// TwinCAT 3 PLC project Tests_and_Samples
// ProgramVersion: 3.1.4023.0
// CompilerDefines: VISU_USEWSTRING
// libraries:
//   Tc2_Standard, * (Beckhoff Automation GmbH)
//   Tc2_System, * (Beckhoff Automation GmbH)
//   Tc3_BAR_Common, * (Beckhoff)
//   Tc3_Module, * (Beckhoff Automation GmbH)
// project tree:
//   / GlobalTextList.TcGTLO, GVL.TcGVL, PlcTask.TcTTO, Visualization Manager.TcVMO (not stored), VISU_TASK.TcTTO
//   GVLs/ Alarms.TcGVL
//   POUs/ AlarmSample.TcPOU, MAIN.TcPOU, TrendSample.TcPOU
//   VISUs/ AlarmsVisSample.TcVIS, TrendsSampleVis.TcVIS, vBrowser.TcVIS, Visualization.TcVIS
//   VISUs/Templates/ tAlarm.TcVIS
// (motion and I/O tree: see PLC project tc3_bar_common)
// real-time tasks:
//   TASK PlcTask: cycle T#10ms, priority 20, ADS port 350
//   TASK VISU_TASK: cycle T#50000us, priority 30, ADS port 351

CONFIGURATION Tests_and_Samples
    RESOURCE PLC ON TwinCAT3
        TASK PlcTask(INTERVAL := T#10ms, PRIORITY := 20);
        TASK VISU_TASK(INTERVAL := T#50000us, PRIORITY := 30);
        PROGRAM MAIN WITH PlcTask : MAIN;
        PROGRAM VisuElems_Visu_Prg WITH VISU_TASK : VisuElems.Visu_Prg;
    END_RESOURCE
END_CONFIGURATION

// ---- GVL.TcGVL
{attribute 'qualified_only'}
VAR_GLOBAL CONSTANT
END_VAR

// ---- GVLs/Alarms.TcGVL
{attribute 'qualified_only'}
VAR_GLOBAL
	SeriosAlarm: FB_Alarm := (AlarmInfo := (AlarmID := "LC224", Color := E_ALarmColors.E_Red, Description := "Серьезная тестовая авария", PossibleCause := "Оператор"));
	NotSeriosAlarm: FB_Alarm := (AlarmType := ALARMTYPE.Alarm_NoQuit, AlarmInfo := (AlarmID := "NQ105", Color := E_ALarmColors.E_Yellow, Description := "Ошибка, которую не нужно квитировать", PossibleCause := "Оператор"));
	SimpleWarning: FB_Alarm := (AlarmType := ALARMTYPE.Alarm_NoQuit, AlarmInfo := (AlarmID := "Wrn01", Color := E_ALarmColors.E_Green, Description := "Событие для записи в журнал", PossibleCause := "Оператор"));
END_VAR

// ---- POUs/MAIN.TcPOU
PROGRAM MAIN
VAR
	bBrowserStart: BOOL;
END_VAR

AlarmSample();// Пример работы с авариями

TrendSample();

END_PROGRAM

// ---- POUs/AlarmSample.TcPOU
PROGRAM AlarmSample
VAR

END_VAR

PRG_Alarms_Core();

END_PROGRAM

// ---- POUs/TrendSample.TcPOU
PROGRAM TrendSample
VAR
	VariableForTrend: REAL;
	t: REAL;
	VariableTrend: FB_TrendChanel := (MinimalValue := -1, MaximalValue := 1);
END_VAR

t:=t+0.01;
VariableForTrend:=SIN(t);
VariableTrend(InputData:= VariableForTrend);

END_PROGRAM

// ---- GlobalTextList.TcGTLO
TEXTLIST GlobalTextList
  789 = '\n\n%s'
  806 = '\n\nАварийное событие'
  101 = ' %s'
  133 = '%s'
  441 = 'PROFIT!?'
  574 = 'Аварийное событие'
  259 = 'История\nаварий'
  733 = 'История аварий'
  97 = 'Квитирование'
  906 = 'Квитирование\n этой аварии'
  227 = 'Квитирование\nвсех аварий'
  328 = 'Квитирование Аварии'
  893 = 'Квитирование этой аварии'
  440 = 'Название'
  618 = 'Название меню'
  740 = 'Пример\nаварий'
  504 = 'Пример\nТрендов'
  550 = 'Пример Аварий'
  641 = 'Пример ещё чего-то'
  12 = 'Пример трендов'
  306 = 'Пример Трендов'
  88 = 'Сброс'
  821 = 'Старт'
  100 = 'Стоп'
  839 = 'Текущие\n аварии'
  126 = 'Текущие\nаварии'
  188 = 'Текущие аварии'
  132 = 'Экран аварий'
END_TEXTLIST

// ---- VISUs/AlarmsVisSample.TcVIS
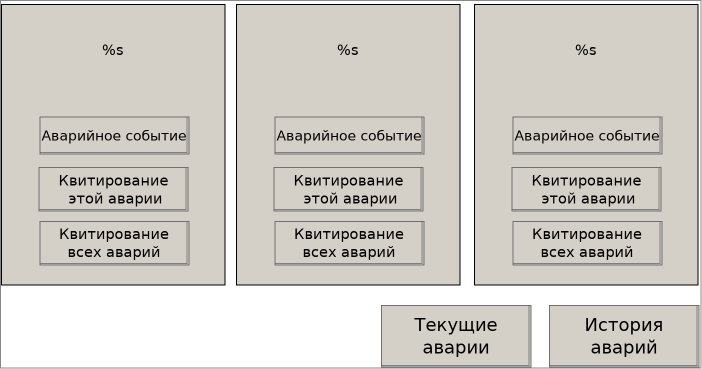
VISUALIZATION AlarmsVisSample  // 702x369
    Frame (1,4 226x283)
        shows tAlarm(alarm := Alarms.SeriosAlarm)
    Frame (236,4 226x283)
        shows tAlarm(alarm := Alarms.NotSeriosAlarm)
    Frame (474,4 226x283)
        shows tAlarm(alarm := Alarms.SimpleWarning)
    Button (381,305 150x62), "Текущие аварии"
        OnMouseClick: OpenDialog Dialog=Tc3_BAR_Common.Current_Alarms_dialog, OpenModal=True, OpenCentered=True
    Button (549,305 150x62), "История аварий"
        OnMouseClick: OpenDialog Dialog=Tc3_BAR_Common.History_Of_Alarms_dialog, OpenModal=True, OpenCentered=True
END_VISUALIZATION

// ---- VISUs/Templates/tAlarm.TcVIS
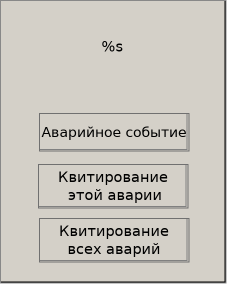
VISUALIZATION tAlarm  // 227x284
VAR_IN_OUT
	alarm: FB_Alarm;
END_VAR
    Rectangle (0,0 225x282), "%s", text variable: alarm.AlarmInfo.Description, colour toggle: Tc3_BAR_Common.LibAlarm.Blink and alarm.isActive
    Button (39,113 150x38), "Аварийное событие"
        toggle alarm.AlarmEvent
    Button (38,164 150x44), "Квитирование этой аварии"
        tap alarm.bQuitAlarm
    Button (39,218 150x44), "Квитирование всех аварий"
        tap Tc3_BAR_Common.LibAlarm.bLocalQuitAllAlarms
END_VISUALIZATION

// ---- VISUs/TrendsSampleVis.TcVIS
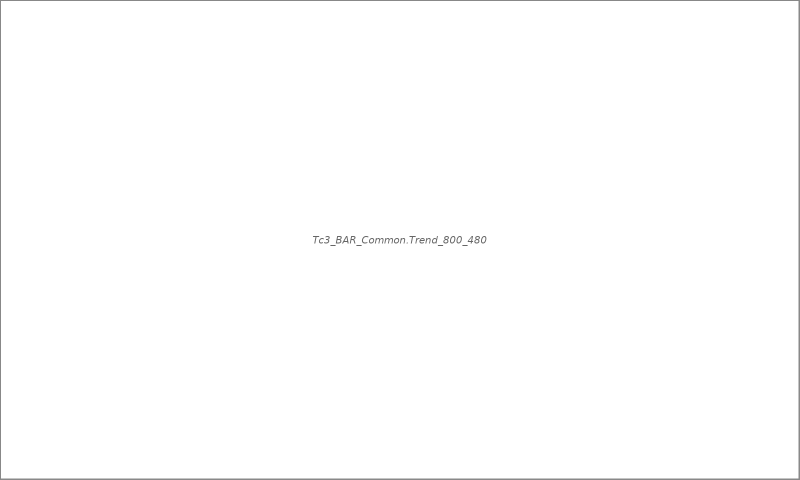
VISUALIZATION TrendsSampleVis  // 800x480
    Frame (0,0 800x480)
        shows Tc3_BAR_Common.Trend_800_480(Header := "Пример названия канала", fb_TrendChanel1 := TrendSample.VariableTrend)
END_VISUALIZATION

// ---- VISUs/vBrowser.TcVIS
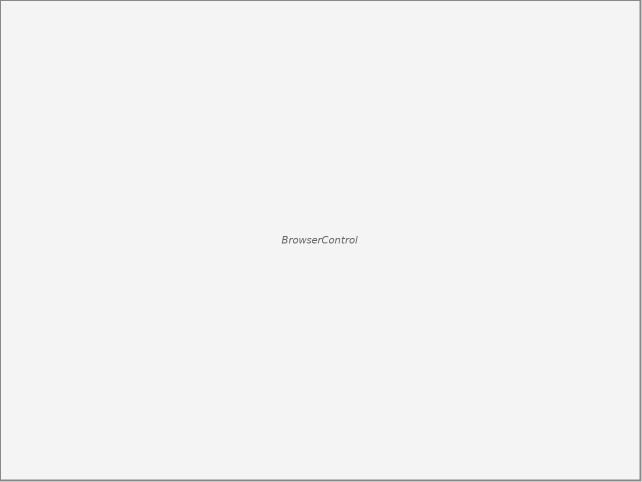
VISUALIZATION vBrowser  // 642x482
    BrowserControl (0,0 640x480)
        p3734058945: 'https://yandex.ru/internet/'
        p2179181546: MAIN.bBrowserStart
END_VISUALIZATION

// ---- VISUs/Visualization.TcVIS
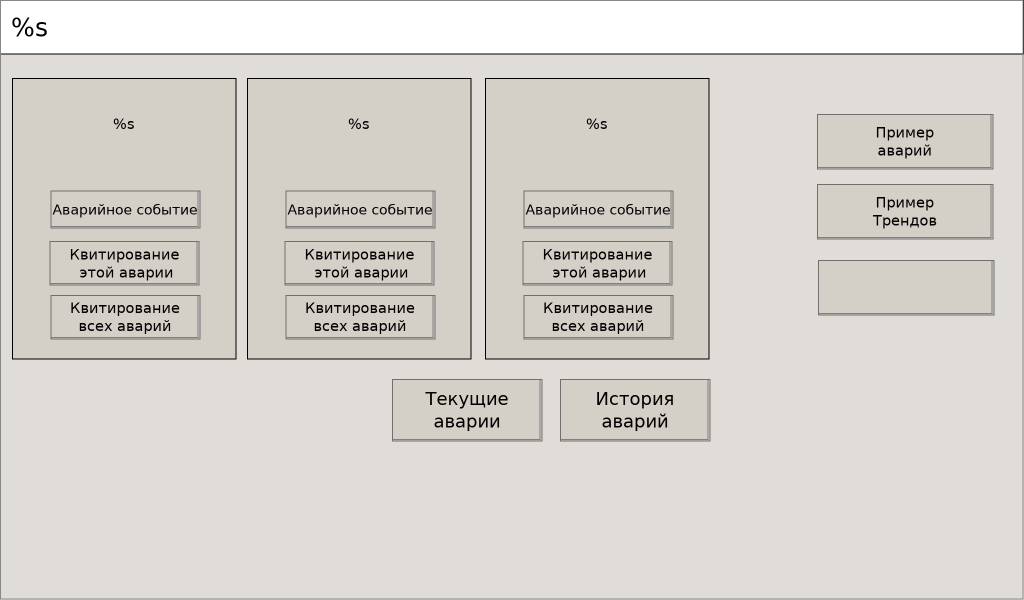
VISUALIZATION Visualization  // 1024x600
    Rectangle (0,0 1024x54), "%s", text variable: Tc3_BAR_Common.LibAlarm.Global_TimeStr
    Frame (11,74 802x474)
        shows AlarmsVisSample()
        shows TrendsSampleVis()
        shows vBrowser()
    Button (817,114 176x55), "Пример аварий"
        OnMouseClick: FrameSelectionChange Selection=SelectedFrame=b3597301-8c91-4ed9-9bbf-06002503f2d3, GlobSel=AssignType=Directly, SelType=Locally
    Button (817,184 176x55), "Пример Трендов"
        OnMouseClick: FrameSelectionChange Selection=SelectedFrame=b3597301-8c91-4ed9-9bbf-06002503f2d3, Selection=1, GlobSel=AssignType=Directly, SelType=Locally
    Button (818,260 176x55)
        OnMouseClick: FrameSelectionChange Selection=SelectedFrame=b3597301-8c91-4ed9-9bbf-06002503f2d3, Selection=2, GlobSel=AssignType=Directly, SelType=Locally
END_VISUALIZATION
